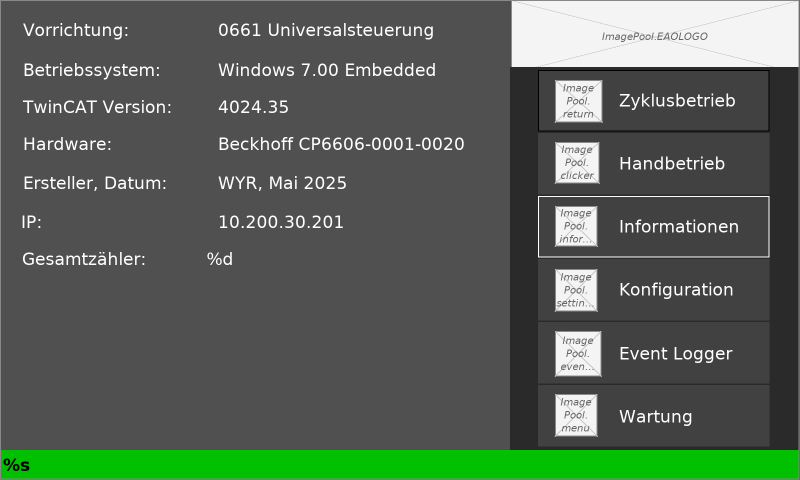
VISUALIZATION Diagnose  // 800x480
    Image (511,0 288x73), image: ImagePool.EAOLOGO
    Rectangle (510,67 289x412)
    Textfield (20,158 177x50), "Ersteller, Datum:"
    Textfield (215,158 288x50), "WYR, Mai 2025"
    Textfield (20,82 177x50), "TwinCAT Version:"
    Textfield (215,82 288x50), "4024.35"
    Textfield (215,45 288x50), "Windows 7.00 Embedded"
    Textfield (20,45 177x50), "Betriebssystem:"
    Textfield (20,5 177x50), "Vorrichtung:"
    Textfield (215,5 288x50), "0661 Universalsteuerung"
    Textfield (20,119 177x50), "Hardware:"
    Textfield (215,119 288x50), "Beckhoff CP6606-0001-0020"
    Textfield (18,197 177x50), "IP:"
    Textfield (215,197 288x50), "10.200.30.201"
    Rectangle (0,450 799x30), "%s", text variable: MAIN.HMI.sStatus, colour variable: MAIN.HMI.nColorInfoBalken
        p3450524324: MAIN.HMI.nColorInfoBalken
    Rectangle (538,70 231x61)
        OnMouseClick: change screen: Zyklusbetrieb
    Textfield (616,70 153x61), "Zyklusbetrieb"
        OnMouseClick: change screen: Zyklusbetrieb
    Rectangle (538,133 231x61)
        OnMouseClick: change screen: Handbetrieb
    Textfield (616,133 153x61), "Handbetrieb"
        OnMouseClick: change screen: Handbetrieb
    Image (555,142 44x41), image: ImagePool.clicker
        OnMouseClick: change screen: Handbetrieb
    Image (555,80 47x42), image: ImagePool.return
        OnMouseClick: change screen: Zyklusbetrieb
    Rectangle (538,196 231x61)
        OnMouseClick: change screen: Diagnose
    Textfield (616,196 153x61), "Informationen"
        OnMouseClick: change screen: Diagnose
    Image (555,206 42x40), image: ImagePool.information
        OnMouseClick: change screen: Diagnose
    Rectangle (538,322 231x61)
        OnMouseClick: change screen: EventLogger
    Textfield (616,323 153x61), "Event Logger"
        OnMouseClick: change screen: EventLogger
    Image (555,331 46x45), image: ImagePool.eventLogger
        OnMouseClick: change screen: EventLogger
    Rectangle (538,259 231x61)
        OnMouseClick: change screen: Konfig1
    Textfield (616,259 153x61), "Konfiguration"
        OnMouseClick: change screen: Konfig1
    Image (555,269 42x42), image: ImagePool.settings
        OnMouseDown: change screen: Konfig1
    Rectangle (538,385 231x61)
        OnMouseClick: change screen: Wartung
    Textfield (616,386 153x61), "Wartung"
        OnMouseClick: change screen: Wartung
    Image (555,394 42x42), image: ImagePool.menu
        OnMouseDown: change screen: Wartung
    Textfield (19,234 477x50), "Gesamtzähler: %d", text variable: MAIN.stStueckzaehler.nGesamt
END_VISUALIZATION

(* stored: Version 1.1.0.1, ProductVersion 3.1.4024.12
   Visu Diagnose: Id {a2bab42d-7dce-4a9b-892c-11236f1ec46e} *)
